(*			
	RafalOS
	Rafał Osajda		20.11.2025		TC 4024.66
	Interfejs przekazywany do modułów tworzących strony
*)
INTERFACE ITF_MCHMIMachineControl_HMI_PrepScr_03_XX

END_INTERFACE

(* stored: Version 1.1.0.1
   Itf ITF_MCHMIMachineControl_HMI_PrepScr_03_XX: Id {4071a637-e5af-0bb1-1f09-4f14060d66c2} *)
